{attribute addProperty BoxType "EK1100-0000-0018"}
{attribute addProperty Id "Beckhoff_EJ2xxxEK1122Beckhoff_EJ2xxxEK1122_7BCCD4D9162A_0001_EJ2008_0000_0017EJ2008_04E0E56B8811A_0002_EJ2008_0000_0018EJ2008_04E0E56B8811A_0003_EJ2128_0000_0016EJ2128_04E0E56B8811A_0004_EJ2502_0000_0023EJ2502_E4940A0412015A_0005_EJ2502_0000_0024EJ2502_E4940A0412015A_0006_EJ2521_0224_0016EJ2521_F54ABF8F36846A_0007_EJ2522_0000_0022EJ2522_E90FBA5F44856A_0008_EJ2809_0000_0017EJ2809_5A2A5F2915219A_0009_EJ2889_0000_0016EJ2889_5A2A5F2915219A_0010_EJ2889_0000_0017EJ2889_5A2A5F2915219"}
{attribute addProperty CRC "2786066703"}
{attribute addProperty SizeInBites "1792"}
{attribute addProperty SizeInBytes "224"}
TYPE Beckhoff_EJ2xxx_A610010F EXTENDS EK1100_179A0949 :
STRUCT
	{attribute addProperty Name "Beckhoff_EJ2xxxEK1122"}
	Beckhoff_EJ2xxxEK1122 : Beckhoff_EJ2xxxEK1122_7BCCD4D9;
	{attribute addProperty Name "A_0001_EJ2008_0000_0017"}
	A_0001_EJ2008_0000_0017 : EJ2008_04E0E56B;
	{attribute addProperty Name "A_0002_EJ2008_0000_0018"}
	A_0002_EJ2008_0000_0018 : EJ2008_04E0E56B;
	{attribute addProperty Name "A_0003_EJ2128_0000_0016"}
	A_0003_EJ2128_0000_0016 : EJ2128_04E0E56B;
	{attribute addProperty Name "A_0004_EJ2502_0000_0023"}
	A_0004_EJ2502_0000_0023 : EJ2502_E4940A04;
	{attribute addProperty Name "A_0005_EJ2502_0000_0024"}
	A_0005_EJ2502_0000_0024 : EJ2502_E4940A04;
	{attribute addProperty Name "A_0006_EJ2521_0224_0016"}
	A_0006_EJ2521_0224_0016 : EJ2521_F54ABF8F;
	{attribute addProperty Name "A_0007_EJ2522_0000_0022"}
	A_0007_EJ2522_0000_0022 : EJ2522_E90FBA5F;
	{attribute addProperty Name "A_0008_EJ2809_0000_0017"}
	A_0008_EJ2809_0000_0017 : EJ2809_5A2A5F29;
	{attribute addProperty Name "A_0009_EJ2889_0000_0016"}
	A_0009_EJ2889_0000_0016 : EJ2889_5A2A5F29;
	{attribute addProperty Name "A_0010_EJ2889_0000_0017"}
	A_0010_EJ2889_0000_0017 : EJ2889_5A2A5F29;
END_STRUCT
END_TYPE

(* stored: Version 1.2.0.0, ProductVersion 3.1.4024.9
   DUT Beckhoff_EJ2xxx_A610010F: Id {df1ce0e6-ece5-43ca-9b25-01c27dfa8e8c} *)
